{attribute 'qualified_only'}
{attribute 'strict'}
TYPE E_LedColor :
(
	Red,
	Green,
	Blue,
	Yellow,
	Cyan,
	Purple,
	White,
	Black
);
END_TYPE

(* stored: Version 1.1.0.1, ProductVersion 3.1.4026.11
   DUT E_LedColor: Id {ad0e60a5-ec28-4c7c-865d-4eb05755c1a3} *)
